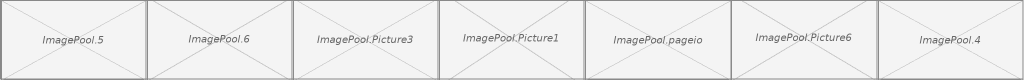
VISUALIZATION N_Footer_Line1  // 1024x80
    Image (878,0 145x80), invisible if: GVL_OF_VU.bVN, input disabled if: GVL_OF_VU.bVN, image: ImagePool.3
        OnMouseDown: ChangeLanguage ChangeLanguage=vn
    Image (878,0 145x80), invisible if: not GVL_OF_VU.bVN, input disabled if: not GVL_OF_VU.bVN, image: ImagePool.4
        OnMouseDown: ChangeLanguage ChangeLanguage=eng
    Image (1,0 145x80), input disabled if: not bResetmanual1, image: ImagePool.5
        OnMouseDown: change screen: MAIN_LINE1
        OnMouseDown: execute {
            MAIN.bModeAuto := TRUE;
            MAIN.bModeManual := FALSE;
            bWriteData := TRUE;
        }
    Image (147,-3 145x84), input disabled if: bResetAuto1, image: ImagePool.6
        OnMouseClick: change screen: N_JarSupply1
        OnMouseClick: execute {
            MAIN.bModeManual := TRUE;
            MAIN.bModeAuto := FALSE;
            bWriteData := TRUE;
        }
    Image (293,-2 145x83), image: ImagePool.Picture3
        OnMouseClick: change screen: N_Setting_Line1
    Image (439,-10 145x96), image: ImagePool.Picture1
        OnMouseClick: change screen: N_Recipe_Line1
    Image (585,0 146x80), image: ImagePool.pageio
        OnMouseClick: change screen: N_PLC_I1
    Image (731,-6 146x87), image: ImagePool.Picture6
        OnMouseClick: change screen: N_Alarm
END_VISUALIZATION

(* stored: Version 1.1.0.1, ProductVersion 3.1.4024.12
   Visu N_Footer_Line1: Id {40442801-519e-4d00-ab8b-8669cfef9af6} *)
